(* CoDeSys 2.3 export: TYPE_LED.EXP *)

(* Data type *)
TYPE Type_LED :
STRUCT
	Switch_ON			:BOOL;
	Switch_RANDOM	:BOOL;
	Config				:Type_LED_CONFIG;
	Brightness			:BYTE;
END_STRUCT
END_TYPE
